// TIA Portal V16 export
// export: Created 2025-05-24T14:07:36.2427825Z, ExportSetting WithDefaults, DisplayName Totally Integrated Automation Portal, DisplayVersion V16, DisplayName TIA Portal Version Control Interface, DisplayVersion V16, DisplayName TIA Portal Openness, DisplayVersion V16, DisplayName STEP 7 Professional, DisplayVersion V16, DisplayName STEP 7 Safety, DisplayVersion V16, DisplayName WinCC Advanced, DisplayVersion V16
FUNCTION "8 - Noodsleutel" : Void   // FC9, LAD
TITLE = Emergency Switch
VERSION : 0.1
// stored: AutoNumber true, IsIECCheckEnabled false, UDAEnableTagReadback false
BEGIN

REGION Network 1
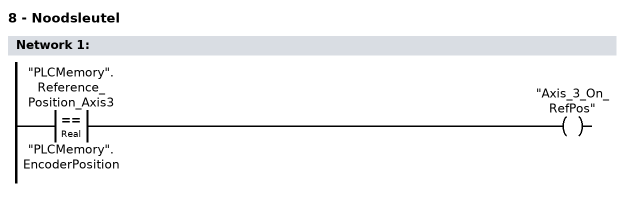
   RUNG wire#powerrail
      { S7_Templates := "SrcType := Real" } EQ_Contact(in1 := "PLCMemory".Reference_Position_Axis3, in2 := "PLCMemory".EncoderPosition)
      Coil( "Axis_3_On_RefPos" )
   END_RUNG
   // the same network as SCL:
   "Axis_3_On_RefPos" := "PLCMemory".Reference_Position_Axis3 = "PLCMemory".EncoderPosition;
END_REGION
END_FUNCTION
